//==================================================================================================
//							Beckhoff Automation Poland
//									19.10.2018
// Program wyświetlający informację o licznikach State Changes i NOT Present - opis ponizej
// Wymagane jest podanie jedynie adresu AMS NET ID Mastera EtherCATa i liczby urzadzen Slave
// State Changes/Not Present
// State Changes - for example if the sync task needs longer then 100ms, state changes from OP to other, but Slave is present
// Not Present - If it switchs back from OP (power off, broken...)
//
//	v1.3 	|| TC v 3.1.4022.25		 	|| - Reset as an input, Presen --> Present 
//	v1.2 	|| TC v 3.1.4022.20		 	|| - Return instruction and some comments
//	v1.1 	|| TC v 3.1.4020.32		 	|| - Dodane wyjscia bOk, bWarning, bError, opisu, zmiana typow zmiennych
//	v1.0 	|| TC v 3.1.4020.32 		|| - Pierwsza wersja
//==================================================================================================
PROGRAM P_EtherCAT_ChangeCounter
VAR CONSTANT
	sAmsNetID_EtherCATMaster				: T_AmsNetId	:= '192.168.40.180.3.1';		// EtherCAT Master AMS Net ID
	wCountOfEtherCATSlaves					: WORD 			:= 67; 							// Count of EtherCAT Slaves
END_VAR
VAR_INPUT
	bReset									: BOOL;
END_VAR
VAR_OUTPUT
	bOK										: BOOL;											// Brak bledow i ostrzezen
	bWarning								: BOOL;											// Ostrzezenie - nie wystepuja w tym podprogramie - wystepuja dla zachowania spojnosci
	bError									: BOOL;											// Zbiorcza flaga bledow
	udiErrorID								: UDINT;
	sErrorDescription						: WSTRING;
END_VAR
VAR
	//======================= State Changes/ ========================
	arrAbnormalStateChangeCounter			: ARRAY [1..wCountOfEtherCATSlaves] OF DWORD; 	// State Changes/  - tablica zawieraca dane dla poszczegilnych Slave
	wAbnormalStateChangeCounterPosition		: WORD;											// Pozycja pierwszego Slavea który zmienił wartosc licznika
	bAbnormalStateChangeCounterChanged		: BOOL;											// Flaga wystapienia zmiany licznika
	//===============================================================
	//======================== /Not Present =========================
	arrPresentStateChangeCounter			: ARRAY [1..wCountOfEtherCATSlaves] OF DWORD; 	// /Not Present  - tablica zawieraca dane dla poszczegilnych Slave
	wPresentStateChangeCounterPosition		: WORD;											// Pozycja pierwszego Slavea który zmienił wartosc licznika
	bPresentStateChangeCounterChanged		: BOOL;											// Flaga wystapienia zmiany licznika
	//===============================================================
	//======================= Internal ==============================
	bFirstCycle								: BOOL := TRUE;
	tonRefresh								: TON;
	tRefreshTime							: TIME := T#200MS;								// Refresh timer
	
	//===============================================================
	//=================== Internal hidden ===========================
	{attribute 'hide'}
	fbADSREAD_AbnormalStateChangeCounter	: ADSREAD;
	{attribute 'hide'}
	fbADSREAD_PresentStateChangeCounter		: ADSREAD;
	//{attribute 'hide'}
	arrAbnormalStateChangeCounterOld		: ARRAY [1..wCountOfEtherCATSlaves] OF DWORD; 	// Stara tablica - do celow porownawczych
	//{attribute 'hide'}
	arrPresenStateChangeCounterOld			: ARRAY [1..wCountOfEtherCATSlaves] OF DWORD; 	// Stara tablica - do celow porownawczych
	{attribute 'hide'}
	i										: WORD;
	{attribute 'hide'}
	ft1										: F_TRIG;
	{attribute 'hide'}
	ft2										: F_TRIG;
	//===============================================================
	rtReset: R_TRIG;
	rtError: R_TRIG;
END_VAR


{region "Is it ready to read?"}
IF sAmsNetID_EtherCATMaster = '' OR wCountOfEtherCATSlaves = 0 THEN
	RETURN;
END_IF
{endregion}
{region "Call FBs"}
// Start reading
tonRefresh(IN:= NOT tonRefresh.Q, PT:= tRefreshTime);

// End of reading 
ft1(CLK:= fbADSREAD_PresentStateChangeCounter.BUSY);
ft2(CLK:= fbADSREAD_AbnormalStateChangeCounter.BUSY);

// Reading
fbADSREAD_PresentStateChangeCounter(
	NETID			:= sAmsNetID_EtherCATMaster,
	PORT			:= 16#FFFF,
	IDXGRP			:= 16#16,
	IDXOFFS			:= 0,
	LEN				:= SIZEOF(arrPresentStateChangeCounter),
	DESTADDR		:= ADR(arrPresentStateChangeCounter),
	READ			:= tonRefresh.Q);

fbADSREAD_AbnormalStateChangeCounter(
	NETID			:= sAmsNetID_EtherCATMaster,
	PORT			:= 16#FFFF,
	IDXGRP			:= 16#13,
	IDXOFFS			:= 0,
	LEN				:= SIZEOF(arrAbnormalStateChangeCounter),
	DESTADDR		:= ADR(arrAbnormalStateChangeCounter),
	READ			:= ft1.Q);
{endregion}
{region "Change detection"}
//================= Checks positon of change ====================
// Check if changed
IF ft1.Q THEN
	IF NOT  bFirstCycle THEN
		FOR i := 1 TO wCountOfEtherCATSlaves DO
			IF arrPresentStateChangeCounter[i] <> arrPresenStateChangeCounterOld[i] THEN
				wPresentStateChangeCounterPosition 		:= i;
				bPresentStateChangeCounterChanged 		:= TRUE;
				EXIT;
			END_IF
		END_FOR
	END_IF
	arrAbnormalStateChangeCounterOld 					:= arrAbnormalStateChangeCounter;
END_IF

IF ft2.Q THEN
	IF NOT  bFirstCycle THEN
		FOR i := 1 TO wCountOfEtherCATSlaves DO
			IF arrAbnormalStateChangeCounter[i] <> arrAbnormalStateChangeCounterOld[i] THEN
				wAbnormalStateChangeCounterPosition 	:= i;
				bAbnormalStateChangeCounterChanged 		:= TRUE;
				EXIT;
			END_IF
		END_FOR
	END_IF
	arrPresenStateChangeCounterOld 						:= arrPresentStateChangeCounter;
	bFirstCycle 										:= FALSE;
END_IF
//===============================================================
{endregion}
{region "Reset and states"}
//  Reset
	 
rtReset(CLK:= bReset);
rtError(CLK:= bError);	
	  
IF rtReset.Q THEN
	wPresentStateChangeCounterPosition 					:= 0;
	wAbnormalStateChangeCounterPosition 				:= 0;
	bPresentStateChangeCounterChanged 					:= FALSE;
	bAbnormalStateChangeCounterChanged 					:= FALSE;
END_IF

// Set outputs
bError 													:= bPresentStateChangeCounterChanged OR bAbnormalStateChangeCounterChanged;
bOK 													:= NOT bError AND NOT bWarning;
	 
IF bError THEN
	udiErrorID											:= 98;
	sErrorDescription									:= "Błąd sterownika | Błąd jednego z urządzeń sieci EtherCAT";
ELSE
	udiErrorID											:= 0;
	sErrorDescription									:= "";		
END_IF	
		   
					
{endregion}

ACTION ACT_SlaveNames:
IF wPresentStateChangeCounterPosition 		= 1 THEN
;
ELSIF wPresentStateChangeCounterPosition 	= 2 THEN
;
ELSIF wPresentStateChangeCounterPosition 	= 3 THEN
;	
ELSIF wPresentStateChangeCounterPosition 	= 4 THEN
;	
ELSIF wPresentStateChangeCounterPosition 	= 5 THEN
;	
END_IF
END_ACTION

END_PROGRAM

(* stored: Version 1.1.0.1, ProductVersion 3.1.4026.13, FileIdentifier a8fae789a9b381e4d48dbd109440737c6e401b87, FileSignature 7548232901ffa1ab40b166722eb22a3ad5ce0d2707c9a6b5711c9b68f7ab752dc504be5152d354e263c30391a633911fca467153c8aadf8d440262391111ad963a2fb4023629ef3ff9c99f96a90555fb68767de6d0feaae72bb0d57480768f46a5f7fb45807afa80c94cc67618d36f078cade72d3eed46e675cfce1fde3b5779d8333d8bf580602196131986489b3c5076e1a8710cf849cb9f281a8943ceeb57af36ac75cf87fe83d15bcb492409d0d5addd91533e93b32e799914938382716ed104aa38ecf5fab86349bf556b259a315b87fa06faf930f79be50d476339925d0cabbb378b6f2721527f90f1d84507676dc10d11fe04983d051af915b38110ee
   POU P_EtherCAT_ChangeCounter: Id {63c50270-9d3e-48fc-b34a-3a1bed7ab1e4}, SpecialFunc None
   Action ACT_SlaveNames: Id {31dfb43e-ddf2-4219-9a64-ff685915632b} *)
